(* IEC 61131-3 sources: ST2CPP/examples/projects/lsp_test, 3 files *)

(* ---- types.st ---- *)
TYPE
    MyPoint :
    STRUCT
        X : INT;
        Y : INT;
    END_STRUCT;

    MyResult :
    STRUCT
        SUM : DINT;
        AVG : DINT;
    END_STRUCT;
END_TYPE

(* ---- utils.st ---- *)
FUNCTION SUM_POINTS : DINT
    VAR_INPUT
        X : INT;
        Y : INT;
    END_VAR
    SUM_POINTS := X + Y;
END_FUNCTION

(* ---- main.st ---- *)
PROGRAM MAIN
    VAR
        P1 : MyPoint;
        P2 : MyPoint;
        Total : DINT;
    END_VAR
    P1.X := 10;
    P1.Y := 20;
    P2.X := P1.X + P1.Y;
    P2.Y := P2.X * 2;
    Total := SUM_POINTS(X := P1.X, Y := P1.Y);
END_PROGRAM
